ABB RobotStudio station: StatieDeRobotTestare.rspag

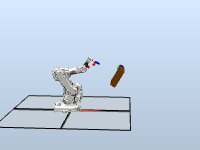
--- station ---
Station StatieDeRobotTestare (saved by RobotStudio 6.4.7206.1027)
Controller System4
  mechanical unit ROB_1: IRB140_6_81_C_03, 6 joints, base frame (0, 0, 0) mm
Layout (positions relative to the parent item):
  - IRB140_6_81_C_03 [mechanism, from Robots\IRB140_6_81_C_G_03.rslib] at (0, 0, 0) mm; joint values [0, -0.6658, 0.4503, 0, -0.8177, 0] (rad or m)
  - Pen [mechanism, from Training Objects\Pen.rslib] at (252.13, 0, 772.19) mm, rotated rx 0 ry 30.8 rz 0 deg
  - Curve_thing [part, from Training Objects\Curve_Thing.rslib] at (820, 200, 750) mm, rotated rx -120 ry 0 rz -90 deg
Attachment: Pen is attached to IRB140_6_81_C_03 / Link6

--- Backups/System4/RAPID/TASK1/PROGMOD/CalibData.mod ---
MODULE CalibData
	PERS tooldata Servo:=[TRUE,[[0,0,114.2],[1,0,0,0]],[0.215,[8.7,12.3,49.2],[1,0,0,0],0.00021,0.00024,0.00009]];
	PERS tooldata Pen_TCP:=[TRUE,[[110,0,140],[0.707106781,0,0.707106781,0]],[1,[10.7435139,0,140],[1,0,0,0],0,0,0]];
    TASK PERS wobjdata canvas1:=[FALSE,TRUE,"",[[0,0,0],[1,0,0,0]],[[820.002,200.001,750.004],[0.353553584,-0.612372324,0.612372324,-0.353553584]]];
ENDMODULE

--- Backups/System4/RAPID/TASK1/PROGMOD/Module1.mod ---
MODULE Module1
    CONST robtarget EXTREME:=[[200.001,126.279387098,-390.936633595],[0.707089442,-0.004951901,0.004951901,0.707089442],[0,0,0,1],[9E+09,9E+09,9E+09,9E+09,9E+09,9E+09]];
    CONST robtarget Target_10:=[[0,0,0],[0.707106781,0,0,0.707106781],[0,-2,1,0],[9E+09,9E+09,9E+09,9E+09,9E+09,9E+09]];
    CONST robtarget Target_20:=[[400,0,0],[0.707106781,0,0,0.707106781],[-1,1,-2,0],[9E+09,9E+09,9E+09,9E+09,9E+09,9E+09]];

    CONST num SHUT_DOWN := -1;
    CONST num TO_WAIT := 0;
    CONST num TO_PAINT := 1;
    CONST num TO_INTRODUCE := 2;

    VAR speeddata drawingSpeed;
    VAR num speedLevel := 0;
    VAR num flag := 0;
    VAR bool repeat := TRUE;

    PERS pos tgPos{500};
    VAR num targetsNum;

    FUNC robtarget create_robtarget(pos position)
       RETURN [position,[0.707106781,0,0,0.707106781],[1,0,0,0],[9E9,9E9,9E9,9E9,9E9,9E9]];
    ENDFUNC

    FUNC speeddata shifting(num base)
        IF base = 0 THEN RETURN v100;
        ELSEIF base = 1 THEN RETURN v300;
        ELSEIF base = 2 THEN RETURN v600;
        ELSE RETURN v1000;
        ENDIF
    ENDFUNC

    ! variable initialization
    FUNC bool init()

        drawingSpeed := shifting(speedLevel);
        targetsNum := 0;
        repeat := TRUE;
        flag := 0;

        RETURN TRUE;

    ENDFUNC

    ! painting process
	PROC EX_PAINT()

        VAR num i := 2;
        drawingSpeed := shifting(speedLevel);

        ! This property is important if targets are created offline/ not in RobotStudio
        ConfL \Off;

        ! Approaching to the canvas is always at maximum speed ( v1000 )
        MoveL create_robtarget(tgPos{1}), shifting(3), z100, Pen_TCP\WObj:=canvas1;
        ! Do while robtarget exists..
        ! This section should be repleaced with for iteration
        WHILE repeat DO

            MoveL create_robtarget(tgPos{i}), drawingSpeed, z100, Pen_TCP\WObj:=canvas1;
            i := i + 1;
            IF i > targetsNum THEN repeat := FALSE; ENDIF

        ENDWHILE

        flag := TO_WAIT;
        repeat := TRUE;
        i := 2;

        ! set the TCP at the starting point
        MoveL EXTREME,shifting(3),z100,Pen_TCP\WObj:=canvas1;

	ENDPROC

    ! other process
    PROC EX_INTRODUCING()

        flag := TO_WAIT;
	ENDPROC

    ! main process
    PROC main()

        IF init() = TRUE THEN

            ! SingArea \Wrist - solvs the 'singularity' problem
            SingArea \Wrist;
            ! set the TCP at the starting point
            MoveL EXTREME,v1000,z100,Pen_TCP\WObj:=canvas1;

            ! A kind of self-made event handler...
            WHILE flag > SHUT_DOWN DO
                IF flag = TO_PAINT THEN EX_PAINT; ENDIF
                IF flag = TO_INTRODUCE THEN EX_INTRODUCING; ENDIF
                WaitTime 0.2;
            ENDWHILE

        ENDIF

    ENDPROC

ENDMODULE

--- Backups/System4/RAPID/TASK1/SYSMOD/LINKEDM.sys ---
%%%
  VERSION:1
  LANGUAGE:ENGLISH
%%%

MODULE LINKEDM (SYSMODULE)

! FOLLOWER
!     Name of electronically linked follower axis used by operator at teach pendent.
      PERS string l_f_axis_name{5}       :=  ["",  "", "", "", ""];

!     Name of the mechanical unit for follower axis.
      PERS string l_f_mecunt_n{5}  :=  ["", "", "", "", ""];

!     Linked follower axis number in the mechanical unit (first axis in mech. unit is number 1).
      PERS num l_f_axis_no{5}      :=  [0,          0,   0,  0,  0];

! MASTER
!     Name of the mechanical unit for linked master axis.
      PERS string l_m_mecunt_n{5} :=  ["", "", "", "", ""];

!     Linked master axis number in the mechanical unit (first axis in mech. unit is number 1).
!     See axis number table in documentation for different master mechanical units.
      PERS num l_m_axis_no{5}     :=  [0,  0,  0,  0,  0];

! POSITION OFFSET
!     The increase of the allowed offset position between the master and follower
!     positions, used when starting AUTO mode. As soon as the offset is decreased
!     the old configurated parameter is used.
!     Example: 3 => the configurated value of allowed offset is increased 3 times.
      PERS num offset_ratio{5}       :=  [10,  10,   10,  10,  10];

! SPEED RATIO
!     Speed_ratio used in AUTO and JOG modes [ very_slow   slow    normal    fast]
!     Value 1 = max allowed manual speed.
      CONST num speed_ratio {20}      := [0.01, 0.01, 0.01, 0.01, 0.01,
                                          0.05, 0.05, 0.05, 0.05, 0.05,
                                          0.20, 0.20, 0.20, 0.20, 0.20,
                                          1.00, 1.00, 1.00, 1.00, 1.00];

! STEP SIZE
!     Displacement position used in JOG mode for each activation of positive or
!     negative movement.                  [very_short    short   normal   long]
!     Unit degees or meter.
      CONST num displacement {20}     := [0.001, 0.001, 0.001, 0.001, 0.001,
                                          0.005, 0.005, 0.005, 0.005, 0.005,
                                          0.020, 0.020, 0.020, 0.020, 0.020,
                                          0.100, 0.100, 0.100, 0.100, 0.100];


!-------------------------------------------------------------
 PROC Linked_m ()
      Linked_m_exe ;
 ENDPROC
ENDMODULE

--- Backups/System4/SYSPAR/EIO.cfg ---
EIO:CFG_1.0:6:1::
#
SYSSIG_IN:

      -Signal "startPainting" -Action "Interrupt" -Arg1 "x" -Arg2 "T_ROB1"\
      -Arg7 "T_ROB1"
#
EIO_SIGNAL:

      -Name "startPainting" -SignalType "DI"
